Fanuc KAREL source: ka00121.KL

-- PROVISIONAL review KL for V1013-1; original PC SHA256 ae0e4857d624b77d7e670b567b5eb797f059e98cf5127faa8bf6e7a21fb2b283
-- Incomplete behavior may be omitted. Consult companion uncertainty JSON. Do not deploy.
PROGRAM KA00121
%NOLOCKGROUP
VAR
  DST : INTEGER
-- UNRESOLVED_DECL SRC type=002018
BEGIN
  -- UNRESOLVED_PC offsets 5-19; opcodes 2E,22,9D,33,B2
  -- UNRESOLVED_PC offsets 24-39; opcodes 22,9D,33,B1,23
  -- UNRESOLVED_PC offsets 44-48; opcodes 7F
END KA00121
